Fanuc KAREL source: ADD_INTPC.kl

PROGRAM T
%NOLOCKGROUP
VAR
 v0 : ARRAY[20] OF BYTE
 v1 : INTEGER
 v2 : INTEGER
 v3 : INTEGER
BEGIN
 ADD_INTPC(v0, v1, v2, v3)
END T
